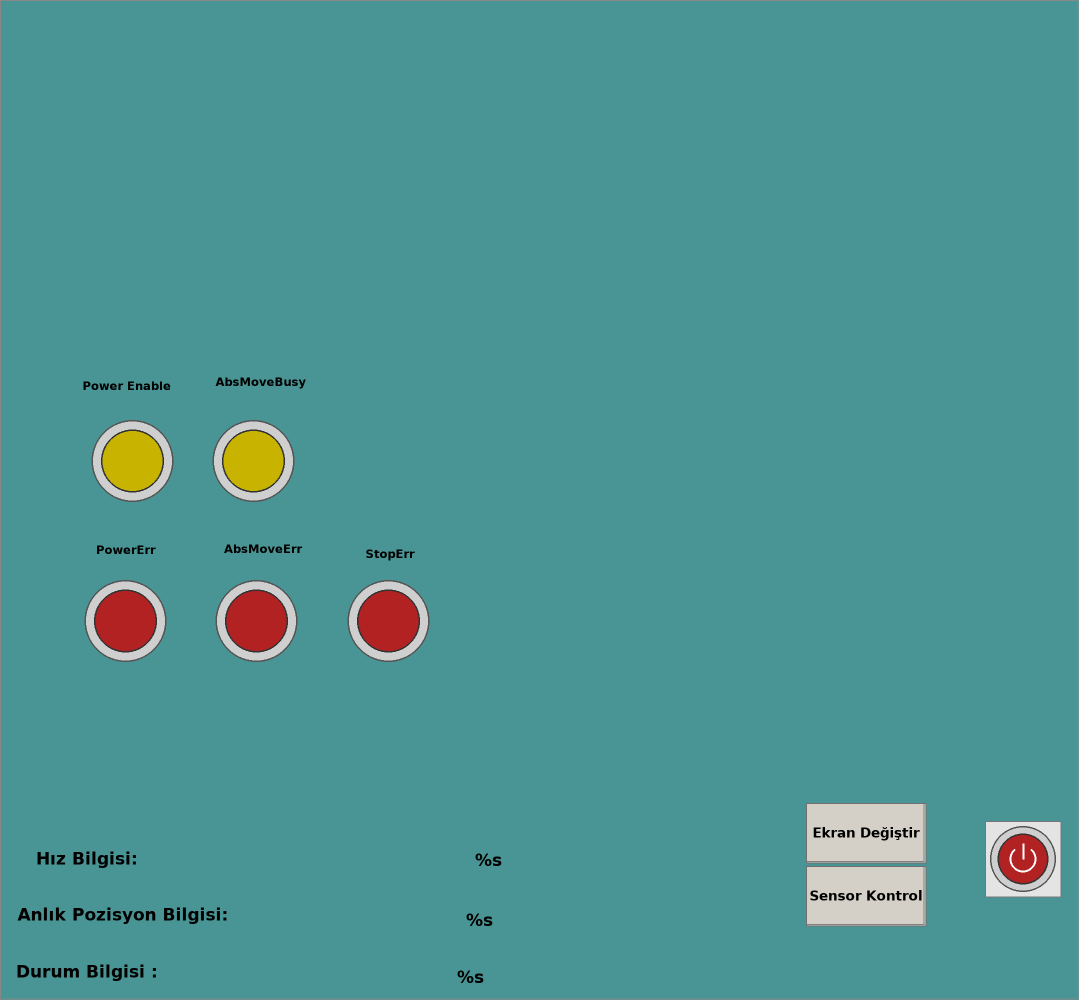
VISUALIZATION VISU_2  // 1079x1000
    Label (3,950 168x43), "Durum Bilgisi :"
    Label (3,893 240x43), "Anlık Pozisyon Bilgisi:"
    Rectangle (240,837 497x46), "%s", text variable: MAIN.sMsgVelo
    Label (3,837 168x43), "Hız Bilgisi:"
    Rectangle (240,897 479x46), "%s", text variable: MAIN.sMsgPosition
    Rectangle (240,954 461x46), "%s", text variable: MAIN.sMsgInfo
    Button (806,803 120x60), "Ekran Değiştir"
        OnMouseClick: change screen: VISU_1
    Button (806,866 120x60), "Sensor Kontrol"
        tap MAIN.bCounter
    PowerSwitch (967,821 112x76), variable: MAIN.bButon, behaviour: TOGGLE, style: Switch-PowerSwitch-Red
    Lamp1 (85,411 95x100), variable: GVL_Axis.stAxis1.OUT.bPowerEnabled, style: Lamp-Lamp1-Yellow
    Lamp1 (206,411 95x100), variable: GVL_Axis.stAxis1.OUT.bMoveAbsBusy, style: Lamp-Lamp1-Yellow
    Lamp1 (78,571 95x100), variable: GVL_Axis.stAxis1.OUT.bPowerErr, style: Lamp-Lamp1-Red
    Lamp1 (209,571 95x100), variable: GVL_Axis.stAxis1.OUT.bMoveAbsErr, style: Lamp-Lamp1-Red
    Lamp1 (341,571 95x100), variable: GVL_Axis.stAxis1.OUT.bStopErr, style: Lamp-Lamp1-Red
    Label (72,372 110x28), "Power Enable"
    Label (206,368 110x28), "AbsMoveBusy"
    Label (335,540 110x28), "StopErr"
    Label (208,535 110x28), "AbsMoveErr"
    Label (71,536 110x28), "PowerErr"
END_VISUALIZATION

(* stored: Version 1.1.0.1, ProductVersion 3.1.4024.4
   Visu VISU_2: Id {9d2947f0-23e8-4c33-9e99-0e6535784a81} *)
